// TIA Portal V18 export
TYPE "LGasp_typePzoListaProfila"
// stored: IsFailsafeCompliant false
   STRUCT
      ID : DInt;   // ID articolo
      "name" : WString[30];   // appoggio nome dell'articolo
      NumeroPezzo : DInt;   // numero del pezzo tagliato
      lenght : LReal := -1.0;   // [mm] - Lunghezza pezzo + sfrido (eventuale)
      cutoffset : LReal := -1.0;   // [mm] - offset foro sincornismo punto di taglio
      wastepiece : Bool;   // TRUE= pezzo di scarto
      info : Struct   // info varie variabili da macchina a macchina
         collo : Int;
         workorder : DInt;
      END_STRUCT;
      options : Array[1..16] of Bool;   // opzioni
      options_str : Array[1..3] of WString[20];   // disponibile per dati specifici dell'impianto
      options_lreal : Array[1..3] of LReal;   // disponibile per dati specifici dell'impianto
      options_dint : Array[1..3] of DInt;   // disponibile per dati specifici dell'impianto
   END_STRUCT;
   // // options[1] : Taglio con ruota metrica (0: No, 1: Si)
   // // options[2] : Articolo rastremato (0: No, 1: Si)
   // // options[3] : Prodotto NON forato (0: pz forato, 1: pz non forato)
   // // options[4] : Taglio con oscuramento (1: abilitato)
   // // options_str[1] : N
END_TYPE
